PROGRAM MAIN
VAR
	
  fbXml : FB_XmlDomParser;
  xmlDoc : SXmlNode;
  xmlConfig : SXmlNode;
  xmlParam : SXmlNode;
  xmlIterator : SXmlIterator;
  xmlParamNode : SXmlNode;
  xmlParamNodeValue : STRING;
  xmlParamNodeADSType : STRING;
  xmlParamNodePath : STRING;
		
	sMessageToParse : STRING(255) := '<Config><Parameter Path="device_1.value" ADSType="DINT">42</Parameter><Parameter Path="device_2.value" ADSType="DINT">24</Parameter></Config>';
	nState : INT := 0;
	
END_VAR



CASE nState OF 

	0 : (* Load XML content *)
			xmlDoc := fbXml.ParseDocument(sMessageToParse);
			nState := nState + 1;
			
	1:
			(* Parse XML nodes *)
			xmlConfig := fbXml.ChildByName(xmlDoc, 'Config');
			xmlIterator := fbXml.Begin(xmlConfig);
			nState := nState + 1;
					
	2:	IF (fbXml.IsEnd(xmlIterator)) THEN 
				nState:= nState +1; 
			ELSE
				xmlParamNode := fbXml.Node(xmlIterator);
  			xmlParamNodePath :=  fbXml.AttributeText(fbXml.Attribute(n:= xmlParamNode, name:='Path'));
  			xmlParamNodeADSType := fbXml.AttributeText(fbXml.Attribute(n:= xmlParamNode, name:='ADSType'));
  			xmlParamNodeValue := fbXml.NodeText(xmlParamNode);	
  			xmlIterator := fbXml.Next(xmlIterator);							
			END_IF
 		
	3:
			xmlIterator := fbXml.End(xmlConfig);
			nState := nState + 1;
			
	4:
			// Error, Done
	
END_CASE

END_PROGRAM

(* stored: Version 1.1.0.1, ProductVersion 3.1.4024.12
   POU MAIN: Id {273e0de6-0218-4241-86c7-fadef2e6f7bb}, SpecialFunc None *)
